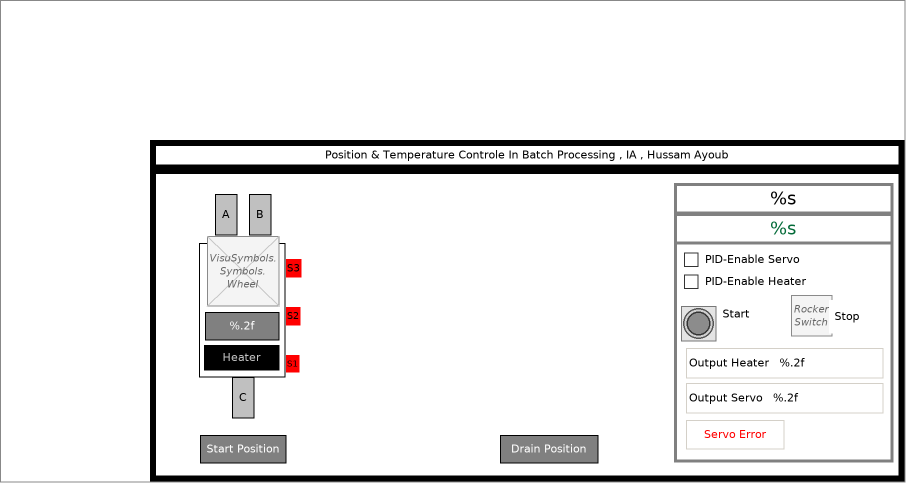
VISUALIZATION UserInterface  // 906x483
    Rectangle (150,168 754x313)
    Rectangle (674,239 219x223)
    Textfield (686,383 197x30), "Output Servo %.2f", text variable: GVL_IO.Output_ServoX
    Textfield (686,348 197x30), "Output Heater %.2f", text variable: GVL_IO.Output_Heater
    Rectangle (200,435 86x28), "Start Position"
    Rectangle (500,435 98x28), "Drain Position"
    Rectangle (199,243 86x134)
        p3560616238: GVL_IO.Output_ServoX * 10
    Textfield (674,213 219x31), "%s", text variable: MAIN.TotalTimeValue
    Checkbox (682,270 123x23), "PID-Enable Heater", variable: MAIN.PID_heater_enable
    Checkbox (682,248 155x23), "PID-Enable Servo", variable: MAIN.PID_Servo_enable
    Textfield (686,420 98x29), "Servo Error", invisible if: NOT GVL_IO.xGenCtrl_Error
    Rectangle (215,194 22x41), "A", colour toggle: GVL_IO.ValveA
    Rectangle (249,194 22x41), "B", colour toggle: GVL_IO.ValveB
    Rectangle (232,377 22x41), "C", colour toggle: GVL_IO.ValveC
        p3560616238: GVL_IO.Output_ServoX * 10
    Rectangle (286,307 14x18), "S2", colour toggle: GVL_IO.Level_S2
        p3560616238: GVL_IO.Output_ServoX * 10
    Rectangle (286,259 15x18), "S3", colour toggle: GVL_IO.Level_S3
        p3560616238: GVL_IO.Output_ServoX * 10
    Rectangle (286,355 13x17), "S1", colour toggle: GVL_IO.Level_S1
        p3560616238: GVL_IO.Output_ServoX * 10
    Image (207,236 72x70), image: VisuSymbols.Symbols.Wheel
        p2858320360: MAIN.Rotation
        p3560616238: GVL_IO.Output_ServoX * 10
    Rectangle (204,345 75x25), "Heater", colour toggle: MAIN.HeaterON
        p3560616238: GVL_IO.Output_ServoX * 10
    RockerSwitch (791,295 41x41), variable: GVL_IO.StopPr, behaviour: TOGGLE, style: Switch-RockerSwitch-Gray
    Textfield (711,299 50x30), "Start"
    Textfield (829,300 36x33), "Stop"
    PushSwitch (681,297 35x53), variable: GVL_IO.StartPr, behaviour: TOGGLE, style: Switch-PushSwitch-Gray
    Textfield (674,183 219x31), "%s", text variable: MAIN.StateString
    Rectangle (150,140 754x30), "Position & Temperature Controle In Batch Processing , IA , Hussam Ayoub"
    Rectangle (205,312 74x28), "%.2f", text variable: GVL_IO.TankLevelSensor
        p3560616238: GVL_IO.Output_ServoX * 10
END_VISUALIZATION

(* stored: Version 1.1.0.1, ProductVersion 3.1.4024.0
   Visu UserInterface: Id {8126f8ab-e6ef-48b6-9ba2-149e11247293} *)
